INTERFACE ITF_AxisControl

METHOD DisableAxis : BOOL
VAR_INPUT
END_VAR
END_METHOD

METHOD EnableAxis : BOOL
VAR_INPUT
END_VAR
END_METHOD

METHOD HaltAxis : BOOL
VAR_INPUT
END_VAR
END_METHOD

METHOD MoveToPosition : BOOL
VAR_INPUT
	Position : MC_LREAL;
	Velocity : MC_LREAL;
END_VAR
END_METHOD

METHOD ResetAxis : BOOL
VAR_INPUT
END_VAR
END_METHOD

END_INTERFACE

(* stored: Version 1.1.0.1
   Itf ITF_AxisControl: Id {67ee2d44-07ee-4a7f-8cf0-2ba796d7942a}
   Method DisableAxis: Id {78e4be45-9441-4dfd-be50-a8de43882816}
   Method EnableAxis: Id {dc495f2e-73cd-4872-9d3b-75cfe930dc9c}
   Method HaltAxis: Id {94883e86-e022-461f-9256-2ce498881fb1}
   Method MoveToPosition: Id {c5eac34c-4010-4d8b-8622-96313c7f08cf}
   Method ResetAxis: Id {fe6c826c-85ca-40eb-8eb2-4dba05c9813a} *)
